(* Logix 5000 project; controller CuteLogix vendor 1 type 14 code 216 rev 30.14; software revision 30.00; part 2 of 2 *)
(* tags used below, declared in another part *)
   AdvancedMath : DINT[10];
   ASCII : STRING[20];
   ASCII_Find : DINT;
   ASCII_Find_Result : DINT;
   ASCII_Qty : DINT;
   ASCII_Start : DINT;
   CmpControl : CONTROL;
   Conv_BCD : DINT[10];
   Dint_Conv : DINT[10];
   For_Index : DINT;
   m_MAFR : MOTION_INSTRUCTION;
   m_MAS : MOTION_INSTRUCTION;
   m_MASD : MOTION_INSTRUCTION;
   m_MASR : MOTION_INSTRUCTION;
   MathConv : REAL[20];
   PID_CV : DINT;
   PID_Inhold : BOOL;
   PID_Inhold_Value : DINT;
   PID_Master : PID;
   PID_PV : DINT;
   PID_Tieback : DINT;
   Real_Conf : REAL[10];
   ResControl : CONTROL;
   Special : DINT[20];
   Special_PID : PID;
   Str_Conv : STRING[10];
   Trig : REAL[20];
   VAxis : AXIS_VIRTUAL;
(* Instructions, continued *)

ROUTINE R021_For_Break   (* ladder *)
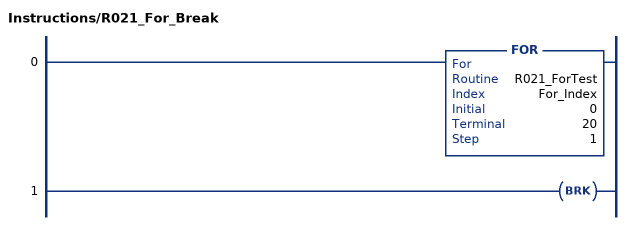
   0: FOR(R021_ForTest,For_Index,0,20,1);
   1: BRK();
END_ROUTINE

ROUTINE R021_ForTest   (* ladder *)
   0: NOP();
END_ROUTINE

ROUTINE R022_Special   (* ladder *)
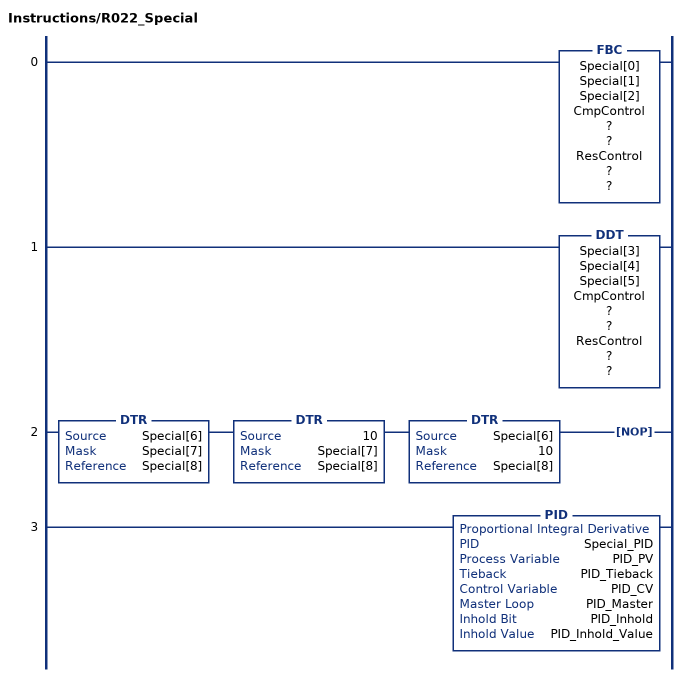
   0: FBC(Special[0],Special[1],Special[2],CmpControl,?,?,ResControl,?,?);
   1: DDT(Special[3],Special[4],Special[5],CmpControl,?,?,ResControl,?,?);
   2: DTR(Special[6],Special[7],Special[8])DTR(10,Special[7],Special[8])DTR(Special[6],10,Special[8])NOP();
   3: PID(Special_PID,PID_PV,PID_Tieback,PID_CV,PID_Master,PID_Inhold,PID_Inhold_Value);
END_ROUTINE

ROUTINE R023_Trig   (* ladder *)
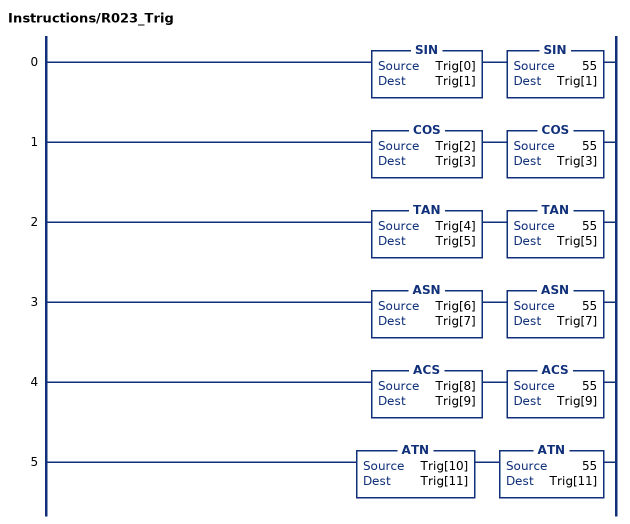
   0: SIN(Trig[0],Trig[1])SIN(55,Trig[1]);
   1: COS(Trig[2],Trig[3])COS(55,Trig[3]);
   2: TAN(Trig[4],Trig[5])TAN(55,Trig[5]);
   3: ASN(Trig[6],Trig[7])ASN(55,Trig[7]);
   4: ACS(Trig[8],Trig[9])ACS(55,Trig[9]);
   5: ATN(Trig[10],Trig[11])ATN(55,Trig[11]);
END_ROUTINE

ROUTINE R024_Advanced_Math   (* ladder *)
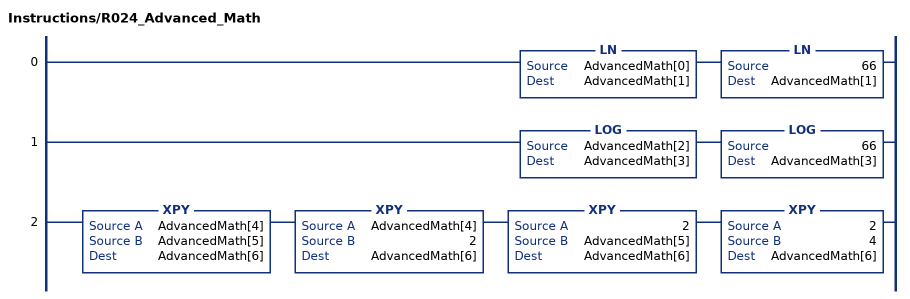
   0: LN(AdvancedMath[0],AdvancedMath[1])LN(66,AdvancedMath[1]);
   1: LOG(AdvancedMath[2],AdvancedMath[3])LOG(66,AdvancedMath[3]);
   2: XPY(AdvancedMath[4],AdvancedMath[5],AdvancedMath[6])XPY(AdvancedMath[4],2,AdvancedMath[6])XPY(2,AdvancedMath[5],AdvancedMath[6])XPY(2,4,AdvancedMath[6]);
END_ROUTINE

ROUTINE R025_Math_Conversion   (* ladder *)
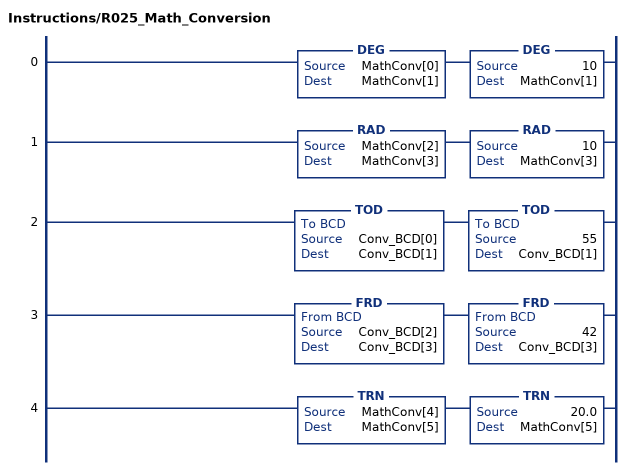
   0: DEG(MathConv[0],MathConv[1])DEG(10,MathConv[1]);
   1: RAD(MathConv[2],MathConv[3])RAD(10,MathConv[3]);
   2: TOD(Conv_BCD[0],Conv_BCD[1])TOD(55,Conv_BCD[1]);
   3: FRD(Conv_BCD[2],Conv_BCD[3])FRD(42,Conv_BCD[3]);
   4: TRN(MathConv[4],MathConv[5])TRN(20.0,MathConv[5]);
END_ROUTINE

ROUTINE R026_Motion_State   (* ladder *)
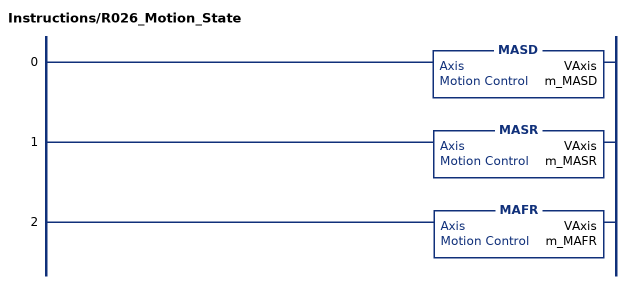
   0: MASD(VAxis,m_MASD);
   1: MASR(VAxis,m_MASR);
   2: MAFR(VAxis,m_MAFR);
END_ROUTINE

ROUTINE R027_Motion_Move   (* ladder *)
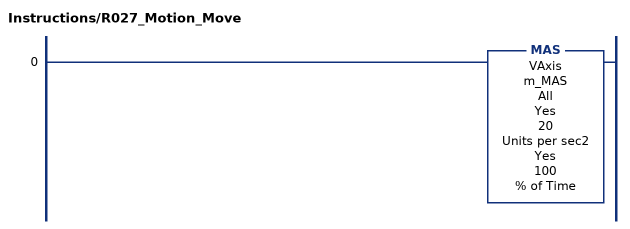
   0: MAS(VAxis,m_MAS,All,Yes,20,Units per sec2,Yes,100,% of Time);
END_ROUTINE

ROUTINE R028_Motion_Group   (* ladder *)
   0: NOP();
END_ROUTINE

ROUTINE R029_Motion_Event   (* ladder *)
   0: NOP();
END_ROUTINE

ROUTINE R030_Motion_Config   (* ladder *)
   0: NOP();
END_ROUTINE

ROUTINE R031_Motion_Coord   (* ladder *)
   0: NOP();
END_ROUTINE

ROUTINE R032_ASCII_String   (* ladder *)
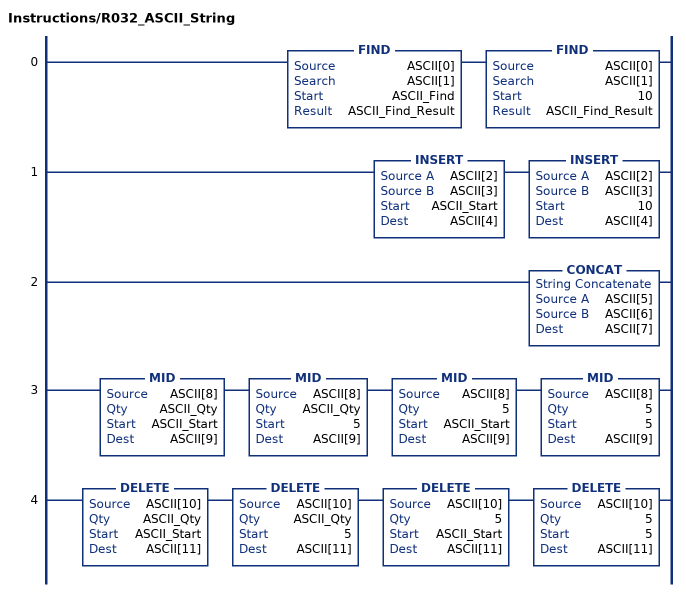
   0: FIND(ASCII[0],ASCII[1],ASCII_Find,ASCII_Find_Result)FIND(ASCII[0],ASCII[1],10,ASCII_Find_Result);
   1: INSERT(ASCII[2],ASCII[3],ASCII_Start,ASCII[4])INSERT(ASCII[2],ASCII[3],10,ASCII[4]);
   2: CONCAT(ASCII[5],ASCII[6],ASCII[7]);
   3: MID(ASCII[8],ASCII_Qty,ASCII_Start,ASCII[9])MID(ASCII[8],ASCII_Qty,5,ASCII[9])MID(ASCII[8],5,ASCII_Start,ASCII[9])MID(ASCII[8],5,5,ASCII[9]);
   4: DELETE(ASCII[10],ASCII_Qty,ASCII_Start,ASCII[11])DELETE(ASCII[10],ASCII_Qty,5,ASCII[11])DELETE(ASCII[10],5,ASCII_Start,ASCII[11])DELETE(ASCII[10],5,5,ASCII[11]);
END_ROUTINE

ROUTINE R033_ASCII_Conv   (* ladder *)
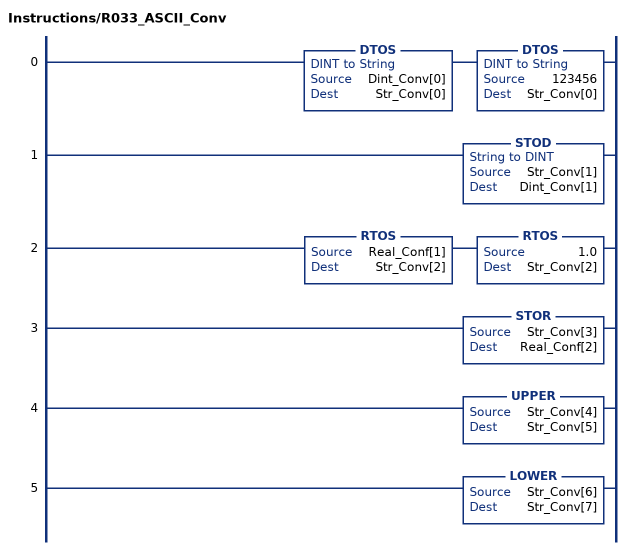
   0: DTOS(Dint_Conv[0],Str_Conv[0])DTOS(123456,Str_Conv[0]);
   1: STOD(Str_Conv[1],Dint_Conv[1]);
   2: RTOS(Real_Conf[1],Str_Conv[2])RTOS(1.0,Str_Conv[2]);
   3: STOR(Str_Conv[3],Real_Conf[2]);
   4: UPPER(Str_Conv[4],Str_Conv[5]);
   5: LOWER(Str_Conv[6],Str_Conv[7]);
END_ROUTINE
END_PROGRAM
